            Step := 10;  
        END_IF

    10:

            fbFileOpen(
                sNetId := '', 
                sPathName := sPath, 
                nMode := FOPEN_MODEAPPEND OR FOPEN_MODETEXT, 
                ePath := PATH_GENERIC, 
                bExecute := TRUE
            );      
        Step := 20;

    20:
        // Czekaj na otwarcie pliku
        fbFileOpen(bExecute := FALSE);
        IF NOT fbFileOpen.bBusy THEN
            IF fbFileOpen.bError THEN
                nErrId := fbFileOpen.nErrId;
                bError := TRUE;
                Step := 500;  
            ELSE
                hFile := fbFileOpen.hFile;
                Step := 300;  
            END_IF
        END_IF 

    300:
        // Zamknij plik
        fbFileClose(
            sNetId := '', 
            hFile := hFile, 
            bExecute := TRUE
        );
        Step := 310;

    310:
        // Czekaj na zamknięcie pliku
        fbFileClose(bExecute := FALSE);
        IF NOT fbFileClose.bBusy THEN
            IF fbFileClose.bError THEN
                nErrId := fbFileClose.nErrId;
                bError := TRUE;
            END_IF
            Step := 500;  
        END_IF

    500:
        bBusy := FALSE;
        Step := 0;
END_CASE

END_PROGRAM

// ---- POUs/DataLogging/P_OEE_Raport.TcPOU
PROGRAM P_OEE_Raport
// Zmienne pomocnicze
VAR
    sCurrentDate        : STRING(10) := '';  // Przechowuje aktualną datę (np. "2023-10-25")
    bNewDay             : BOOL := FALSE;     // Flaga wskazująca, że rozpoczął się nowy dzień
    hFile               : UINT := 0;        // Uchwyt pliku
    sFilePath           : T_MaxString := ''; // Ścieżka do pliku
    nBytesToWrite       : UDINT := 0;        // Liczba bajtów do zapisania
    sLineToWrite             : T_MaxString := ''; // Bufor na dane do zapisania
    dtString            : STRING(20) := '';  // Czas zmiany w formacie tekstowym
    fbFileSeek          : FB_FileSeek;       // Blok do pozycjonowania wskaźnika pliku
    fbFileTell          : FB_FileTell;       // Blok do odczytu pozycji wskaźnika pliku
    fbFileGets          : FB_FileGets;       // Blok do odczytu linii z pliku
    bFileIsEmpty        : BOOL := FALSE;     // Flaga wskazująca, czy plik jest pusty
	RisingEdge			:R_trig;
	bSaveManuel			:BOOL;
	Step				:INT;
	bBusy 				:BOOL;
	bError				:BOOL;
	nErrId				:UDINT;
	nIndex				:INT;
	sFolderPath: STRING(255) := 'C:\OEE\';
	fbFileOpen: FB_FileOpen;
    fbFileWrite: FB_FileWrite;
    fbFileClose: FB_FileClose;
	b10step:BOOL;
	rtrig10MinsWork :r_trig;
	tonworkfor10min	:TON;
	AStBadPackageReasonText :ARRAY[0..63] OF S_Information_Text;
    i : INT;
    aIdToName: ARRAY[11..24] OF WSTRING := [
        "Wadliwa butelka lub proces przerwany:","Waga za mała:","Waga za duża:",
        "Brak odłożenia platynki:", "Platynka źle położona:", "Platynka nie zgrzana:",
        "Brak nas.(Słomka):", "Brak nasadki za zakręcarkami:","Brak nasadki przed zakręcarką:",
        "Nie zakręcono zakręcarką szczękową:", "Nasadka źle zakręcona:", "ROPP nie nałożony", 
		"ROPP nie zakręcony","ROPP brak za stacją"];
	bWork10min: BOOL;
	tontimerforevery10min :ton;
END_VAR

// Główna logika
IF Step=0 THEN
	bError:=FALSE;
END_IF
rtrig10MinsWork(CLK:=P_ADS_OEE.btonDelayAfterStart);
tonworkfor10min(in:=bWork10min, PT:=T#5M);
tontimerforevery10min(in:=NOT bWork10min AND P_ADS_OEE.btonDelayAfterStart, PT:=T#5M);
IF rtrig10MinsWork.Q  OR bSaveManuel OR tontimerforevery10min.q THEN
	bWork10min:=TRUE;
END_IF
IF tonworkfor10min.Q THEN
	bWork10min:=FALSE;
END_IF
RisingEdge(CLK := bSaveManuel OR tonworkfor10min.q OR P_ADS_OEE.bCycleReset OR P_ADS_OEE.btonConfectionEnding);

IF rtrig10MinsWork.Q  OR RisingEdge.q THEN 
	FOR i := 0 TO 63 DO
	    IF (P_ADS_OEE.AStBadPackageReason[i].udiID >= 11) AND (P_ADS_OEE.AStBadPackageReason[i].udiID <= 24) THEN
	        AStBadPackageReasonText[i].desc := aIdToName[P_ADS_OEE.AStBadPackageReason[i].udiID];
	    ELSE
	        AStBadPackageReasonText[i].desc := "";
	    END_IF;
	   
	    AStBadPackageReasonText[i].wsDescription := P_ADS_OEE.AStBadPackageReason[i].wsDescription;
	END_FOR;
END_IF

CASE Step OF
    0:
        // Sprawdź, czy zmienił się dzień
        IF LEFT(WSTRING_TO_STRING(P_time.s_time_mainscreen), 10) <> sCurrentDate THEN
            sCurrentDate := LEFT(WSTRING_TO_STRING(P_time.s_time_mainscreen), 10);  // Zaktualizuj datę
            bNewDay := TRUE;  // Ustaw flagę nowego dnia
        END_IF

        // Jeśli wystąpiło zdarzenie zapisu lub zmiany receptury
        IF RisingEdge.Q THEN
            bBusy := TRUE;
            bError := FALSE;
            nErrId := 0;
            nIndex := 0;

            // Utwórz ścieżkę do pliku na podstawie aktualnej daty
            sFilePath := CONCAT(sFolderPath, 'OEE_Raport_');
            sFilePath := CONCAT(sFilePath, sCurrentDate);
            sFilePath := CONCAT(sFilePath, '.csv');

            Step := 10;  // Przejdź do kroku otwarcia pliku
        END_IF

    10:
        // Otwórz plik
        IF bNewDay THEN
            // Jeśli nowy dzień, otwórz plik w trybie zapisu (tworzy nowy plik)
            fbFileOpen(
                sNetId := '', 
                sPathName := sFilePath, 
                nMode := FOPEN_MODEWRITE OR FOPEN_MODETEXT, 
                ePath := PATH_GENERIC, 
                bExecute := TRUE
            );
            b10step := TRUE;
        ELSE
            // Jeśli stary dzień, otwórz plik w trybie dopisywania
            fbFileOpen(
                sNetId := '', 
                sPathName := sFilePath, 
                nMode := FOPEN_MODEAPPEND OR FOPEN_MODETEXT, 
                ePath := PATH_GENERIC, 
                bExecute := TRUE
            );
            b10step := TRUE;
        END_IF
        Step := 20;

    20:
        // Czekaj na otwarcie pliku
        fbFileOpen(bExecute := FALSE);
        IF NOT fbFileOpen.bBusy THEN
            IF fbFileOpen.bError THEN
                nErrId := fbFileOpen.nErrId;
                bError := TRUE;
                Step := 500;  // Przejdź do kroku obsługi błędów
            ELSE
                hFile := fbFileOpen.hFile;
                Step := 30;  // Przejdź do kroku weryfikacji pliku
            END_IF
        END_IF

    30:
        // Sprawdź, czy plik jest pusty (tylko dla nowego dnia)
        IF bNewDay THEN
            fbFileTell(
                sNetId := '', 
                hFile := hFile, 
                bExecute := TRUE
            );
            Step := 35;
        ELSE
            Step := 40;  // Pomijaj weryfikację dla starego dnia
        END_IF

    35:
        // Czekaj na odczyt pozycji wskaźnika pliku
        fbFileTell(bExecute := FALSE);
        IF NOT fbFileTell.bBusy THEN
            IF fbFileTell.nSeekPos = 0 THEN
                bFileIsEmpty := TRUE;  // Plik jest pusty
            ELSE
                bFileIsEmpty := FALSE; // Plik nie jest pusty
            END_IF
            Step := 40;
        END_IF

    40:
        // Przygotuj dane do zapisu
        IF NOT fbFileTell.bBusy THEN
            sLineToWrite := CONCAT(WSTRING_TO_STRING(P_time.s_time_mainscreen), '|');
			sLineToWrite := CONCAT(sLineToWrite, WSTRING_TO_STRING(gvl_recipe.s_recipe_name));
            sLineToWrite := CONCAT(sLineToWrite, '|');
			sLineToWrite := CONCAT(sLineToWrite, INT_TO_STRING(REAL_TO_INT(P_ADS_OEE.uiCounterBadBottles)));
			sLineToWrite := CONCAT(sLineToWrite, '|');
            sLineToWrite := CONCAT(sLineToWrite, INT_TO_STRING(REAL_TO_INT(P_ADS_OEE.uiCounterGoodBottles)));
			sLineToWrite := CONCAT(sLineToWrite, '|');
			sLineToWrite := CONCAT(sLineToWrite, WSTRING_TO_STRING(AStBadPackageReasonText[0].desc));
            sLineToWrite := CONCAT(sLineToWrite, ':');
            sLineToWrite := CONCAT(sLineToWrite, WSTRING_TO_STRING(AStBadPackageReasonText[0].wsDescription));
			sLineToWrite := CONCAT(sLineToWrite, '|');			
            sLineToWrite := CONCAT(sLineToWrite, WSTRING_TO_STRING(AStBadPackageReasonText[1].desc));
            sLineToWrite := CONCAT(sLineToWrite, ':');
            sLineToWrite := CONCAT(sLineToWrite, WSTRING_TO_STRING(AStBadPackageReasonText[1].wsDescription));
			sLineToWrite := CONCAT(sLineToWrite, '|');
			sLineToWrite := CONCAT(sLineToWrite, WSTRING_TO_STRING(AStBadPackageReasonText[2].desc));
            sLineToWrite := CONCAT(sLineToWrite, ':');                                     
            sLineToWrite := CONCAT(sLineToWrite, WSTRING_TO_STRING(AStBadPackageReasonText[2].wsDescription));
			sLineToWrite := CONCAT(sLineToWrite, '|');
			sLineToWrite := CONCAT(sLineToWrite, WSTRING_TO_STRING(AStBadPackageReasonText[3].desc));
            sLineToWrite := CONCAT(sLineToWrite, ':');
            sLineToWrite := CONCAT(sLineToWrite, WSTRING_TO_STRING(AStBadPackageReasonText[3].wsDescription));
			sLineToWrite := CONCAT(sLineToWrite, '|');
			sLineToWrite := CONCAT(sLineToWrite, WSTRING_TO_STRING(AStBadPackageReasonText[4].desc));
            sLineToWrite := CONCAT(sLineToWrite, ':');
            sLineToWrite := CONCAT(sLineToWrite, WSTRING_TO_STRING(AStBadPackageReasonText[4].wsDescription));
			sLineToWrite := CONCAT(sLineToWrite, '|');
			sLineToWrite := CONCAT(sLineToWrite, WSTRING_TO_STRING(AStBadPackageReasonText[5].desc));
            sLineToWrite := CONCAT(sLineToWrite, ':');
            sLineToWrite := CONCAT(sLineToWrite, WSTRING_TO_STRING(AStBadPackageReasonText[5].wsDescription));
			sLineToWrite := CONCAT(sLineToWrite, '|');
			sLineToWrite := CONCAT(sLineToWrite, WSTRING_TO_STRING(AStBadPackageReasonText[6].desc));
            sLineToWrite := CONCAT(sLineToWrite, ':');
            sLineToWrite := CONCAT(sLineToWrite, WSTRING_TO_STRING(AStBadPackageReasonText[6].wsDescription));
			sLineToWrite := CONCAT(sLineToWrite, '|');
			sLineToWrite := CONCAT(sLineToWrite, WSTRING_TO_STRING(AStBadPackageReasonText[7].desc));
            sLineToWrite := CONCAT(sLineToWrite, ':');
            sLineToWrite := CONCAT(sLineToWrite, WSTRING_TO_STRING(AStBadPackageReasonText[7].wsDescription));
			sLineToWrite := CONCAT(sLineToWrite, '|');
			sLineToWrite := CONCAT(sLineToWrite, WSTRING_TO_STRING(AStBadPackageReasonText[8].desc));
            sLineToWrite := CONCAT(sLineToWrite, ':');
            sLineToWrite := CONCAT(sLineToWrite, WSTRING_TO_STRING(AStBadPackageReasonText[8].wsDescription));
			sLineToWrite := CONCAT(sLineToWrite, '|');
			sLineToWrite := CONCAT(sLineToWrite, WSTRING_TO_STRING(AStBadPackageReasonText[9].desc));
            sLineToWrite := CONCAT(sLineToWrite, ':');
            sLineToWrite := CONCAT(sLineToWrite, WSTRING_TO_STRING(AStBadPackageReasonText[9].wsDescription));
			sLineToWrite := CONCAT(sLineToWrite, '|');
			sLineToWrite := CONCAT(sLineToWrite, WSTRING_TO_STRING(AStBadPackageReasonText[10].desc));
            sLineToWrite := CONCAT(sLineToWrite, ':');
            sLineToWrite := CONCAT(sLineToWrite, WSTRING_TO_STRING(AStBadPackageReasonText[10].wsDescription));
			sLineToWrite := CONCAT(sLineToWrite, '|');
			sLineToWrite := CONCAT(sLineToWrite, WSTRING_TO_STRING(AStBadPackageReasonText[11].desc));
            sLineToWrite := CONCAT(sLineToWrite, ':');
            sLineToWrite := CONCAT(sLineToWrite, WSTRING_TO_STRING(AStBadPackageReasonText[11].wsDescription));
			sLineToWrite := CONCAT(sLineToWrite, '|');
			sLineToWrite := CONCAT(sLineToWrite, WSTRING_TO_STRING(AStBadPackageReasonText[12].desc));
            sLineToWrite := CONCAT(sLineToWrite, ':');
            sLineToWrite := CONCAT(sLineToWrite, WSTRING_TO_STRING(AStBadPackageReasonText[12].wsDescription));
			sLineToWrite := CONCAT(sLineToWrite, '|');
			sLineToWrite := CONCAT(sLineToWrite, WSTRING_TO_STRING(AStBadPackageReasonText[13].desc));
            sLineToWrite := CONCAT(sLineToWrite, ':');
            sLineToWrite := CONCAT(sLineToWrite, WSTRING_TO_STRING(AStBadPackageReasonText[13].wsDescription));
			sLineToWrite := CONCAT(sLineToWrite, '|');
			sLineToWrite := CONCAT(sLineToWrite, 'Czas pracy(min):');
			sLineToWrite := CONCAT(sLineToWrite, UINT_TO_STRING(P_ADS_OEE.udiCounterExecuteTime));
			sLineToWrite := CONCAT(sLineToWrite, '$N');

            nBytesToWrite := LEN(sLineToWrite);

            // Zapisz dane do pliku
            fbFileWrite(
                sNetId := '', 
                hFile := hFile, 
                pWriteBuff := ADR(sLineToWrite), 
                cbWriteLen := nBytesToWrite, 
                bExecute := TRUE
            );
            Step := 50;
        ELSE
            Step := 300;  // Przejdź do kroku zamknięcia pliku
        END_IF

    50:
        // Czekaj na zakończenie zapisu
        fbFileWrite(bExecute := FALSE);
        IF NOT fbFileWrite.bBusy THEN
            IF fbFileWrite.bError THEN
                nErrId := fbFileWrite.nErrId;
                bError := TRUE;
                Step := 500;  // Przejdź do kroku obsługi błędów
            ELSE
                Step := 300;  // Przejdź do kroku zamknięcia pliku po jednokrotnym zapisie
            END_IF
        END_IF

    300:
        // Zamknij plik
        fbFileClose(
            sNetId := '', 
            hFile := hFile, 
            bExecute := TRUE
        );
        Step := 310;

    310:
        // Czekaj na zamknięcie pliku
        fbFileClose(bExecute := FALSE);
        IF NOT fbFileClose.bBusy THEN
            IF fbFileClose.bError THEN
                nErrId := fbFileClose.nErrId;
                bError := TRUE;
            END_IF
            Step := 500;  // Przejdź do kroku obsługi błędów
        END_IF

    500:
        // Zakończ procedurę
        bBusy := FALSE;
        bNewDay := FALSE;  // Zresetuj flagę nowego dnia
        Step := 0;
END_CASE

END_PROGRAM

// ---- POUs/ADS/P_ADS_OEE.TcPOU
PROGRAM P_ADS_OEE
VAR
	btonDelayAfterStart :BOOL;
	fbRead_1: FB_ReadAdsSymByName;	
	fbCyclicReadout: TON;
	uiCounterGoodBottles :UINT;
	fbRead_2: FB_ReadAdsSymByName;
	AStBadPackageReason  :ARRAY[0..63] OF S_Information;
	fbRead_3: FB_ReadAdsSymByName;
	uiCounterBadBottles  :UINT;
	fbRead_4: FB_ReadAdsSymByName;
	fbRead_5: FB_ReadAdsSymByName;
	bCycleReset :BOOL;
	udiCounterExecuteTime :UINT;
	fbRead_6: FB_ReadAdsSymByName;
	btonConfectionEnding:BOOL;
	fbRead_7: FB_ReadAdsSymByName;
	
END_VAR

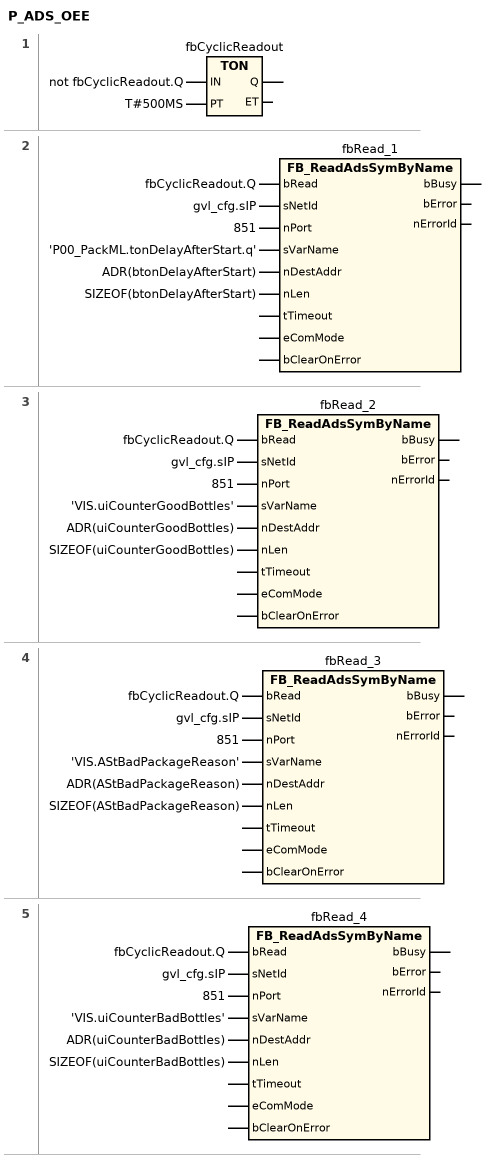
// NETWORK 1
fbCyclicReadout(IN := not fbCyclicReadout.Q, PT := T#500MS); // TON

// NETWORK 2
fbRead_1(
    bRead := fbCyclicReadout.Q,
    sNetId := gvl_cfg.sIP,
    nPort := 851,
    sVarName := 'P00_PackML.tonDelayAfterStart.q',
    nDestAddr := ADR(btonDelayAfterStart),
    nLen := SIZEOF(btonDelayAfterStart)); // FB_ReadAdsSymByName

// NETWORK 3
fbRead_2(
    bRead := fbCyclicReadout.Q,
    sNetId := gvl_cfg.sIP,
    nPort := 851,
    sVarName := 'VIS.uiCounterGoodBottles',
    nDestAddr := ADR(uiCounterGoodBottles),
    nLen := SIZEOF(uiCounterGoodBottles)); // FB_ReadAdsSymByName

// NETWORK 4
fbRead_3(
    bRead := fbCyclicReadout.Q,
    sNetId := gvl_cfg.sIP,
    nPort := 851,
    sVarName := 'VIS.AStBadPackageReason',
    nDestAddr := ADR(AStBadPackageReason),
    nLen := SIZEOF(AStBadPackageReason)); // FB_ReadAdsSymByName

// NETWORK 5
fbRead_4(
    bRead := fbCyclicReadout.Q,
    sNetId := gvl_cfg.sIP,
    nPort := 851,
    sVarName := 'VIS.uiCounterBadBottles',
    nDestAddr := ADR(uiCounterBadBottles),
    nLen := SIZEOF(uiCounterBadBottles)); // FB_ReadAdsSymByName

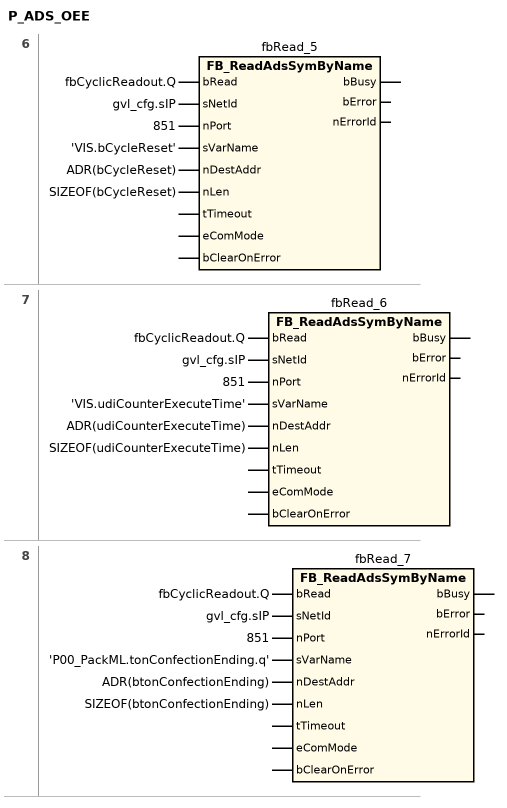
// NETWORK 6
fbRead_5(
    bRead := fbCyclicReadout.Q,
    sNetId := gvl_cfg.sIP,
    nPort := 851,
    sVarName := 'VIS.bCycleReset',
    nDestAddr := ADR(bCycleReset),
    nLen := SIZEOF(bCycleReset)); // FB_ReadAdsSymByName

// NETWORK 7
fbRead_6(
    bRead := fbCyclicReadout.Q,
    sNetId := gvl_cfg.sIP,
    nPort := 851,
    sVarName := 'VIS.udiCounterExecuteTime',
    nDestAddr := ADR(udiCounterExecuteTime),
    nLen := SIZEOF(udiCounterExecuteTime)); // FB_ReadAdsSymByName

// NETWORK 8
fbRead_7(
    bRead := fbCyclicReadout.Q,
    sNetId := gvl_cfg.sIP,
    nPort := 851,
    sVarName := 'P00_PackML.tonConfectionEnding.q',
    nDestAddr := ADR(btonConfectionEnding),
    nLen := SIZEOF(btonConfectionEnding)); // FB_ReadAdsSymByName

END_PROGRAM

// ---- POUs/Persistent/P_PersistentDataSave.TcPOU
PROGRAM P_PersistentDataSave
VAR
	fbSaveChanges :FB_Save;
	sFolderPath: STRING(255) := 'C:\Recipe_changes\';
END_VAR

IF P_persistent.bWritePersistent THEN
	fbSaveChanges.sFilePath := CONCAT(sFolderPath, 'Recipe_change');
    fbSaveChanges.sFilePath := CONCAT(fbSaveChanges.sFilePath, p_24h_C1_2.sCurrentDate);
    fbSaveChanges.sFilePath := CONCAT(fbSaveChanges.sFilePath, '.csv');
	fbSaveChanges();
END_IF

END_PROGRAM

// ---- FB/FB_Save.TcPOU
//-----------------------------------------------------------------------------------------------------
//																
//									 	Tkmatik sp z o.o.
//
//	Name					:		FB_Save
//	Author					:		AM
//	Release Date			:		12.01.2022
//	Current ver				:		v 0.1
// 	Last correction 		:		12.01.2022
// 
//	Description				:
//		Special FB for saving structures to BINARY files						
//
//	Requared hardware		:
//
// 	Configuration			:
//
//
//-----------------------------------------------------------------------------------------------------

FUNCTION_BLOCK FB_Save
VAR_INPUT
	sFilePath											:	STRING(255);					//	File path (e.g. 'C:\1.txt'
	pStructAdr											:	PVOID;                          //	Pointer on data struct
	udiStructSize										:	UDINT;                          //	Size of datastruct
	bExecute											:	BOOL;                           //
END_VAR                                                                                     
VAR_OUTPUT                                                                                  
	bBusy												:	BOOL;                           //	FB is Busy
	bDone												:	BOOL;                           //	Load cycle done, DATA actual 
	bError												:	BOOL;                           //	Flag error
	nErrId												:	UDINT;                          //	Error ID
END_VAR                                                                                     
VAR                                                                                         
	fbFileOpen											:	FB_FileOpen;                    //	FB for opening 
	fbFileClose											:	FB_FileClose;                   //	FB for closing
	fbFileWrite											:	FB_FileWrite;                   //	FB for saving
	hFile												:	UINT;                           //	File hendler
	eMainCase											:	E_FileOpSteps;                  //	Main cycle case value
	rtExecute											:	R_TRIG;                         //	Rtrig for start
END_VAR

ACT_FBs();
ACT_Main();

ACTION ACT_FBs:
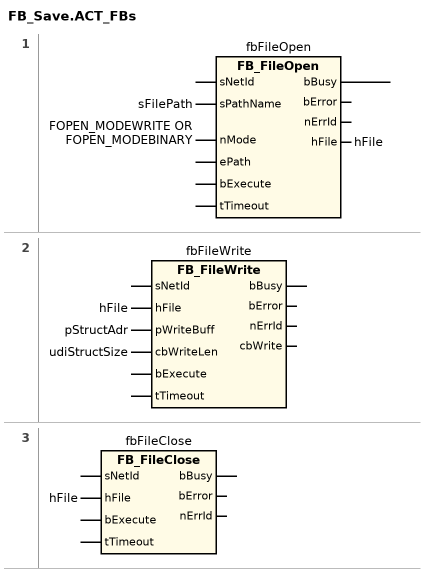
// NETWORK 1
fbFileOpen(sPathName := sFilePath, nMode := FOPEN_MODEWRITE OR FOPEN_MODEBINARY, hFile => hFile); // FB_FileOpen

// NETWORK 2
fbFileWrite(hFile := hFile, pWriteBuff := pStructAdr, cbWriteLen := udiStructSize); // FB_FileWrite

// NETWORK 3
fbFileClose(hFile := hFile); // FB_FileClose
END_ACTION

ACTION ACT_Main:
rtExecute(CLK:=bExecute);
IF (NOT bExecute) THEN
	bDone												:=	FALSE;
END_IF

CASE eMainCase OF
	E_FileOpSteps.eNop:
		fbFileClose.bExecute							:=	FALSE;
		fbFileOpen.bExecute								:=	FALSE;
		fbFileWrite.bExecute							:=	FALSE;
		bBusy											:=	FALSE;
		
		IF (rtExecute.Q) THEN
			bError										:=	FALSE;
			nErrId										:=	0;
			eMainCase									:=	E_FileOpSteps.eStartOpen;
			bBusy										:=	TRUE;
		END_IF
		
	E_FileOpSteps.eStartOpen:
		fbFileOpen.bExecute								:=	TRUE;
		eMainCase										:=	E_FileOpSteps.eWaitOpen;

	E_FileOpSteps.eWaitOpen:
		IF (fbFileOpen.bError) THEN
			bError										:=	TRUE;
			nErrId										:=	10;
			eMainCase									:=	E_FileOpSteps.eNop;
		END_IF
		IF (NOT fbFileOpen.bBusy) THEN
			fbFileOpen.bExecute							:=	FALSE;
			eMainCase									:=	E_FileOpSteps.eStartOper;
		END_IF
		
	E_FileOpSteps.eStartOper:
		fbFileWrite.bExecute							:=	TRUE;
		eMainCase										:=	E_FileOpSteps.eWaitOper;
		
	E_FileOpSteps.eWaitOper:
		IF (fbFileWrite.bError) THEN
			bError										:=	TRUE;
			nErrId										:=	20;
			eMainCase									:=	E_FileOpSteps.eNop;
		END_IF
		IF (NOT fbFileWrite.bBusy) THEN
			fbFileWrite.bExecute						:=	FALSE;
			eMainCase									:=	E_FileOpSteps.eStartClose;
		END_IF
		
	E_FileOpSteps.eStartClose:
		fbFileClose.bExecute							:=	TRUE;
		eMainCase										:=	E_FileOpSteps.eWaitClose;
	
	E_FileOpSteps.eWaitClose:
		IF (fbFileClose.bError) THEN
			bError										:=	TRUE;
			nErrId										:=	30;
			eMainCase									:=	E_FileOpSteps.eNop;
		END_IF
		IF (NOT fbFileClose.bBusy) THEN
			fbFileClose.bExecute						:=	FALSE;
			bDone										:=	TRUE;
			eMainCase									:=	E_FileOpSteps.eNop;
		END_IF	
		
END_CASE
END_ACTION

END_FUNCTION_BLOCK

// ---- POUs/Persistent/P_Persistent.TcPOU
//==================================================================================================
//							Beckhoff Automation Poland
//									25.04.2018
//		Program obslugujacy pamiec nieulotna 
//	v1.4    || TC v 3.1.4026.19		|| - Obsługa UPS
// 	v1.3	|| TC v 3.1.4022.16		|| - Przeniesienie logowania do EvenLogger'a do programu P_SystemDiag_EventLog
// 	v1.2	|| TC v 3.1.4022.0		|| - Dodanie akcji UPS
//	v1.1 	|| TC v 3.1.4020.14 	|| - Dodane wyjscia bOk, bWarning, bError
//	v1.0 	|| TC v 3.1.4020.0 		|| - Pierwsza wersja
//==================================================================================================
PROGRAM P_Persistent
VAR_INPUT
	sAmsNetID_EtherCATMaster	: T_AmsNetId	:= '192.168.40.160.3.1';			// EtherCAT Master AMS Net ID
	bWritePersistent			: BOOL;
	bReset						: BOOL;
END_VAR
VAR_OUTPUT
	bOK							: BOOL 						:= TRUE;				// Brak bledow i ostrzezen
	bWarning					: BOOL;												// Ostrzezenie
	bError						: BOOL;												// Zbiorcza flaga bledow
	udiErrorID					: UDINT;
	sErrorDescription			: WSTRING;
	bWrited						: BOOL;
	bPowerFailDetect			: BOOL;
END_VAR
VAR																			
	iStep						: INT;
	fbWritePersistentData		: FB_WritePersistentData;
	
	//fbUPS						: FB_S_UPS;
	//fbUPS_CB3011				: FB_S_UPS_CB3011;
	//fbUPS_CX51x0				: FB_S_UPS_CX51x0;
	//fbUPS_CX9020_U900			: FB_S_UPS_CX9020_U900;
	//fbUPS_BAPI					: FB_S_UPS_BAPI;
	fbUPS_CU8130				:FB_GetUPSStatus;
	
	//eUpsMode					: E_S_UPS_Mode;
	//eUpsState					: E_S_UPS_State;
	
	
	iNumberOfWrites				: INT;
	rtWritePersistent			: R_TRIG;
END_VAR


ACT_UPS();
ACT_WritePersistent();

fbUPS_CU8130.stStatus.ePowerStatus;
fbUPS_CU8130.stStatus.eBatteryStatus;
fbUPS_CU8130.stStatus.nPowerFailCnt;
fbUPS_CU8130.stStatus.eCommStatus;
IF fbUPS_CU8130.stStatus.ePowerStatus=2 AND NOT bWrited THEN
	bWritePersistent:=TRUE;
ELSE
	bWritePersistent:=FALSE;
END_IF

ACTION ACT_UPS:
//fbUPS_CX9020_U900
//(
//	sNetID							:= sAmsNetID_EtherCATMaster, 
//	iPLCPort						:= 851, 
//	tTimeout						:= DEFAULT_ADS_TIMEOUT, 
//	eUpsMode						:= E_S_UPS_Mode.eSUPS_WrPersistData_Shutdown,
//	ePersistentMode					:= E_PersistentMode.SPDM_2PASS, 
//	tRecoverTime					:= T#10S, 
//	bPowerFailDetect				=> bPowerFailDetect, 
//	eState							=> eUpsState
//);


//fbUPS_CX51x0
//(
//	sNetID							:= sAmsNetID_EtherCATMaster, 
//	iPLCPort						:= 851, 
//	iUPSPort						:= 16#588, 
//	tTimeout						:= DEFAULT_ADS_TIMEOUT, 
//	eUpsMode						:= E_S_UPS_Mode.eSUPS_WrPersistData_Shutdown, 
//	ePersistentMode					:= E_PersistentMode.SPDM_2PASS, 
//	tRecoverTime					:= T#10S, 
//	bPowerFailDetect				=> bPowerFailDetect, 
//	eState							=> eUpsState
//);
fbUPS_CU8130
(	sNetID							:='192.168.40.180.1.1',
	nPort							:=851,
	bEnable							:=TRUE,
	bValid							=>,
	bError	=>,
	nErrId =>,
	stStatus =>,);
END_ACTION

ACTION ACT_WritePersistent:
rtWritePersistent(CLK:= bWritePersistent);


CASE iStep OF

0:
	IF rtWritePersistent.Q THEN
		fbWritePersistentData.PORT												:= _AppInfo.AdsPort;
		fbWritePersistentData.MODE												:= SPDM_2PASS;	
		fbWritePersistentData.START												:= TRUE;
		bWrited																	:= FALSE;
		iStep:= 10;
	END_IF

10:
	IF NOT fbWritePersistentData.BUSY THEN
		IF NOT fbWritePersistentData.ERR THEN
			fbWritePersistentData.START											:= FALSE;
			bWrited																:= TRUE;	
			iNumberOfWrites														:= iNumberOfWrites + 1;
			iStep:= 20;
		END_IF
	END_IF

	IF fbWritePersistentData.ERR THEN
 	
		bWrited																	:= FALSE;
		bError																	:= TRUE;	
		udiErrorID																:= fbWritePersistentData.ERRID;
		sErrorDescription														:= "Błąd zapisu zmiennych PERSISTENT";
		iStep:= 900;
	END_IF
	
20:
	IF NOT bWritePersistent THEN
		iStep:= 0;
	END_IF	
	
900:
	bOK																			:= FALSE;
	
	IF bReset THEN
		fbWritePersistentData.START												:= FALSE;
	END_IF
	IF NOT bReset THEN
		fbWritePersistentData.START												:= TRUE;
	END_IF
	
	
	IF NOT fbWritePersistentData.BUSY THEN
		IF NOT fbWritePersistentData.ERR THEN 
			bOK																	:= TRUE;
			bError																:= FALSE;
			udiErrorID															:= 0;
			sErrorDescription													:= "";
			iStep:= 0;	
		END_IF
	END_IF
	

END_CASE


fbWritePersistentData();
END_ACTION

END_PROGRAM

// ---- FB/FB_Persistent.TcPOU
FUNCTION_BLOCK FB_Persistent

(********************************************************************************************************)
(*								Beckhoff Automation Poland												*)
(* 									FB_Persistent 	v1.5												*)
(* 										20.08.2014														*)
(* 							v1.5 - zmiana minimalnego interwalu zapisu									*)
(* 					Blok funkcyjny zapisujący zmienne typu persistent na karcie CF						*)
(* 						Możliwy zapis na żądanie lub z określoną częstotliwością.  						*)
(* 				Pozostawienie wejscia tInterval bez zmiennej wyłacza funkcję zapisu cyklicznego			*)
(* 							Minimalny czas między zapisem cyklicznym 30s								*)
(* 				Konieczne jest dodanie biblioteki TcUtilities.lib, TcSystem.lib oraz TcBase.lib			*)
(*			 UWAGA: Blok przygotowany dla RunTime 1 port 851 - typowa konfiguracja 						*)
(*______________________________________________________________________________________________________*)

VAR_INPUT
	bWrite					: BOOL;						(*Zapis na rozkaz *)
	tInterval				: TIME:=T#71582M47S295MS;	(*Czestotliwosc zapisu na karte CF*)
END_VAR
VAR_OUTPUT
	bBusy					: BOOL;
	bErr					: BOOL;
	udErrID					: UDINT;
END_VAR
VAR
	fbWritePersistentData	: FB_WritePersistentData; 	(* Blok zapisu *)
	t1						: TON;						(* Timer zapisu *)
	_GETCURTASKINDEX		: GETCURTASKINDEX;			(* Informacja o Tasku *)
	BIndex					: BYTE;						(* Nr tasku *)
END_VAR

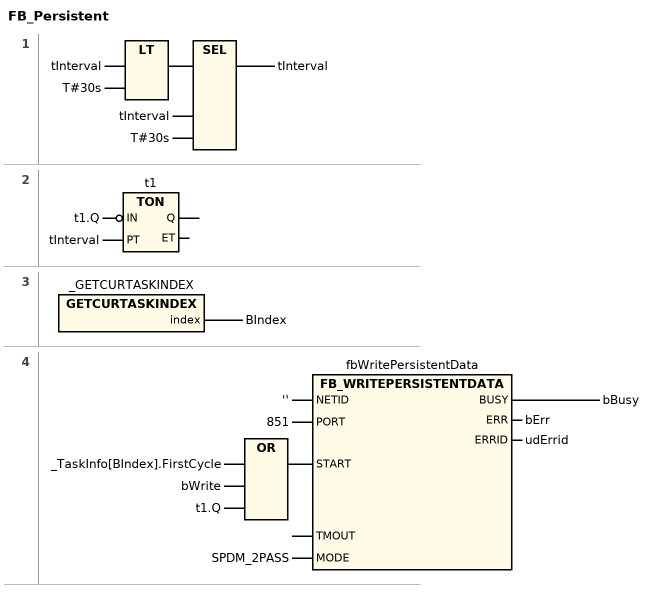
// NETWORK 1
tInterval := SEL(tInterval < T#30s, tInterval, T#30s);

// NETWORK 2
t1(IN := NOT t1.Q, PT := tInterval); // TON

// NETWORK 3
_GETCURTASKINDEX(); // GETCURTASKINDEX
BIndex := _GETCURTASKINDEX.index;

// NETWORK 4
fbWritePersistentData(
    NETID := '',
    PORT := 851,
    START := _TaskInfo[BIndex].FirstCycle OR bWrite OR t1.Q,
    MODE := SPDM_2PASS,
    ERR => bErr,
    ERRID => udErrid); // FB_WRITEPERSISTENTDATA
bBusy := fbWritePersistentData.BUSY;

END_FUNCTION_BLOCK

// ---- FB/FB_ReadWriteLogCSV.TcPOU
(*
Nazwa:			FB_ReadWriteCSV
Opis:			Zapis uzytkownikow do pliku CSV
Wersja:			v0.1
Data:			2018-10-31
Autor:			
Urzadzenia:		
Konfiguracja:	
Info:
*)
FUNCTION_BLOCK FB_ReadWriteLogCSV
VAR
	sCSVLine				: T_MaxString := '';(* Single CSV text line (row, record), we are using string as record buffer (your are able to see read fields)  *)
	sCSVField				: T_MaxString := '';(* Single CSV field value (column, record field) *)
	nRow	 				: UDINT 	:= 0;(* Row number (record) *)
	nColumn					: UDINT 	:= 0;(* Column number (record field) *)
	hFile					: UINT		:= 0;(* File handle of the source file *)
	step					: DWORD 	:= 0;
	fbFileOpen				: FB_FileOpen;(* Opens file *)
	fbFileClose				: FB_FileClose;(* Closes file *)
	fbFileGets				: FB_FileGets;(* Reads one record (line) *)
	fbReader				: FB_CSVMemBufferReader;(* Helper function block used to parse CSV data bytes (single record line) *)
	fbFilePuts				: FB_FilePuts;(* Writes one record (line) *)
	fbWriter				: FB_CSVMemBufferWriter;(* Helper function block used to create CSV data bytes (single record line) *)
	database				: ARRAY[0..239, 0..10] OF STRING(100);(* Target PLC database *)
	i						: INT;
	iNum					: INT;
	BusyFTRIG				: F_TRIG;	// Zakonczenie zapisu/odczytu pliku
	CommandRTRIG			: R_TRIG;	// Wykrycie zapisu/odczytu
	ErrorFileDataUsers		: R_TRIG;	// Błąd zapisu/odczytu
	bNewFile				: BOOL;		// Utworzenie nowego pliku
	iMode					: INT;		// Zapis/odczyt
	
	MAX_CSV_ROWS 			: UDINT := 239;
	MAX_CSV_COLUMNS 		: UDINT := 10;
	MAX_CSV_FIELD_LENGTH	: UDINT := 100;
	
//	fbGetDateTime			: NT_GetTime;
	sDateTime				: STRING[200];
	fbFileTell				: FB_FileTell;
	fbEOF					: FB_EOF;
	fbFileSeek				: FB_FileSeek;
	
	sLineToWrite			:STRING(255);
END_VAR
	
VAR_INPUT
	bRead					: BOOL;		//Sygnal odczytu pliku
	bWrite					: BOOL;		//Sygnal zapisu pliku
	stDataArray				: ARRAY [0..239] OF S_LogData;	//Tablica z danymi
	sNetId					: T_AmsNetId := '';	(* TwinCAT system network address *)
	sFileName				: T_MaxString ;(* CSV destination file path and name *)
END_VAR
VAR_OUTPUT
	bError					: BOOL;		// Sygnal błedu
	bBusy					: BOOL;		// Sygnal zajetosci
	bDone					: BOOL;		// Sygnal zakonczenia odczytu/zapisu
	nErrId					: UDINT;	// Numer bledu
END_VAR

CASE step OF
	0:	(* Wait for rising edge at bWrite variable *)
		IF bWrite (*AND NOT fbGetDateTime.BUSY*) THEN
			bWrite 		:= FALSE;
			bBusy 		:= TRUE;
			bError		:= FALSE;
			nErrId		:= 0;
			hFile		:= 0;
			nRow	 	:= 1;			//było 0
			nColumn		:= 0;
			step 		:= 1;
			//wybiera elementy do zapisania
			FOR iNum := 0 TO TO_INT(MAX_CSV_ROWS) DO
//				sDateTime			:=SYSTEMTIME_TO_STRING(fbGetDateTime.TIMESTR);
//				sDateTime			:=DELETE(sDateTime,11,1);	//Usuwa datę
//				sDateTime			:=LEFT(sDateTime,find(sDateTime,'.')-1); //usuwa licznik ms
				    


				//	sLineToWrite := CONCAT(WSTRING_TO_STRING(P_time.s_time_mainscreen), ',');
   		 		//	sLineToWrite := CONCAT(sLineToWrite, REAL_TO_STRING(P_ADS_SCREW.lrGripperScrewer1TorqueCV));
   		 		//	sLineToWrite := CONCAT(sLineToWrite, ',');
   		 		//	sLineToWrite := CONCAT(sLineToWrite, WSTRING_TO_STRING(gvl_recipe.s_recipe_name));
   		 		//	sLineToWrite := CONCAT(sLineToWrite, '$N');	




				database[iNum,0]		:= WSTRING_TO_STRING(P_time.s_time_mainscreen);
				database[iNum,1]		:= REAL_TO_STRING(stDataArray[iNum].arData[0]);
				database[iNum,2]		:= REAL_TO_STRING(stDataArray[iNum].arData[1]);
				database[iNum,3]		:= REAL_TO_STRING(stDataArray[iNum].arData[2]);
				database[iNum,4]		:= REAL_TO_STRING(stDataArray[iNum].arData[3]);
				database[iNum,5]		:= REAL_TO_STRING(stDataArray[iNum].arData[4]);
				database[iNum,6]		:= REAL_TO_STRING(stDataArray[iNum].arData[5]);
				database[iNum,7]		:= REAL_TO_STRING(stDataArray[iNum].arData[6]);
				database[iNum,8]		:= REAL_TO_STRING(stDataArray[iNum].arData[7]);
				database[iNum,9]		:= REAL_TO_STRING(stDataArray[iNum].arData[8]);
				database[iNum,10]		:= REAL_TO_STRING(stDataArray[iNum].arData[9]);
				
//				database[iNum,0]		:= GVL.arLogDataSave1[iNum].tTime;
//				database[iNum,1]		:= REAL_TO_STRING(GVL.arLogDataSave1[iNum].arData[0]);
//				database[iNum,2]		:= REAL_TO_STRING(GVL.arLogDataSave1[iNum].arData[1]);
//				database[iNum,3]		:= REAL_TO_STRING(GVL.arLogDataSave1[iNum].arData[2]);
//				database[iNum,4]		:= REAL_TO_STRING(GVL.arLogDataSave1[iNum].arData[3]);
//				database[iNum,5]		:= REAL_TO_STRING(GVL.arLogDataSave1[iNum].arData[4]);
//				database[iNum,6]		:= REAL_TO_STRING(GVL.arLogDataSave1[iNum].arData[5]);
//				database[iNum,7]		:= REAL_TO_STRING(GVL.arLogDataSave1[iNum].arData[6]);
//				database[iNum,8]		:= REAL_TO_STRING(GVL.arLogDataSave1[iNum].arData[7]);
//				database[iNum,9]		:= REAL_TO_STRING(GVL.arLogDataSave1[iNum].arData[8]);
//				database[iNum,10]		:= REAL_TO_STRING(GVL.arLogDataSave1[iNum].arData[9]);
			END_FOR
			//zmienia . na , żeby szybciej przetwarzać dane w excelu
//			FOR i:=1 TO UDINT_TO_INT(MAX_CSV_COLUMNS) BY 1 DO
//				database[1,i]:=REPLACE(database[1,i],',',1,FIND(database[1,i],'.'));
//			END_FOR
		END_IF
	1:	(* Open source file *)
		fbFileOpen(bExecute := FALSE);
		fbFiletell(bExecute := FALSE);	//potrzebne do wykrycia nowego pliku
	//	fbEOF(bExecute:=FALSE);
		fbFileSeek(bExecute:=FALSE);	//potrzebne do wykrycia nowego pliku
		fbFileOpen( 	sNetId := sNetId, sPathName := sFileName, nMode := FOPEN_MODEAPPEND OR FOPEN_MODETEXT,(* Open file in TEXT mode! *)
						ePath := PATH_GENERIC, bExecute := TRUE );
		step := 2;
	2:(* Wait until open not busy *)
		fbFileOpen( bExecute := FALSE, bError => bError, nErrID => nErrID, hFile => hFile );
		
		IF NOT fbFileOpen.bBusy THEN
			IF NOT fbFileOpen.bError THEN
				//step := 3;
				//sprawdź czy to nowy plik czy dopisujesz
				//próbuje cofnąć pointer odczytu o -2
				fbFileSeek(sNetId := sNetId,eOrigin := SEEK_END, nSeekPos:=-2, hFile := hFile, bExecute:= TRUE, tTimeout:=T#2S);
				IF NOT fbFileSeek.bBusy THEN
					//sprawdzam gdzie jest pointer
					fbFileTell(sNetId := sNetId, hFile := hFile, bExecute:= TRUE, tTimeout:=T#2S);
					IF NOT fbFileTell.bBusy THEN
						step := 3;
						//jak pointer = 0 to znaczy że zapisano nowy plik - dodaj nagłówki do Excela
						IF fbFileTell.nSeekPos = 0 THEN
							database[1,0]		:='Czas';
							database[1,1]		:= GVL_Screw.arDataLogScrew[0];
							database[1,2]		:= GVL_Screw.arDataLogScrew[1];
							database[1,3]		:= GVL_Screw.arDataLogScrew[2];
							database[1,4]		:= GVL_Screw.arDataLogScrew[3];
							database[1,5]		:= GVL_Screw.arDataLogScrew[4];
							database[1,6]		:= GVL_Screw.arDataLogScrew[5];
							database[1,7]		:= GVL_Screw.arDataLogScrew[6];
							database[1,8]		:= GVL_Screw.arDataLogScrew[7];
							database[1,9]		:= GVL_Screw.arDataLogScrew[8];
							database[1,10]		:= GVL_Screw.arDataLogScrew[9];
						END_IF
					END_IF
				END_IF
			ELSE(* Error: file not found? *)
				step := 100;
			END_IF
		END_IF
	3:(* Convert one PLC record to CSV format *)
		sCSVLine := '';
		fbWriter.eCmd := eEnumCmd_First;(* Write first field value *)
		IF nRow <= MAX_CSV_ROWS THEN
			FOR nColumn := 0 TO MAX_CSV_COLUMNS BY 1 DO
				sCSVField := STRING_TO_CSVFIELD( database[ nRow, nColumn ], FALSE );(* TODO: Get field value from your application *)
				(* Add new field to the record buffer *)
				fbWriter( 	pBuffer := ADR( sCSVLine ), cbBuffer := SIZEOF( sCSVLine ) - 1, putValue := sCSVField, pValue := 0, cbValue := 0,
							bCRLF := ( nColumn = MAX_CSV_COLUMNS ) );(* bCRLF == TRUE => Write CRLF after the last field value *)
				IF fbWriter.bOk THEN
					fbWriter.eCmd := eEnumCmd_Next;(* Write next field value *)
				ELSE(* Error *)
					step := 100;
					RETURN;
				END_IF
			END_FOR(* FOR nColumn := 0... *)
			(* FB_FilePuts adds allready CR (carriage return) to the written line.
			We have to replace the $R$L characters with $L character to avoid double CR. *)
			IF RIGHT( sCSVLine, 2 ) = '$R$L' THEN
				sCSVLine := REPLACE( sCSVLine, '$L', 2, LEN( sCSVLine ) - 1 );
			END_IF
			nRow := nRow + 1;(* Increment number of created records (rows) *)
			step := 4;(* Write record to the file *)
		ELSE(* All rows written => Close file *)
			step := 10;
		END_IF
	4:	(* Write single text line *)
		fbFilePuts( bExecute := FALSE );
		fbFilePuts( sNetId := sNetId, hFile := hFile, sLine := sCSVLine, bExecute := TRUE );
		step := 5;
	5:(* Wait until write not busy *)
		fbFilePuts( bExecute := FALSE, bError => bError, nErrID => nErrID );
		IF NOT fbFilePuts.bBusy THEN
			IF NOT fbFilePuts.bError THEN
				step := 3;(* Write next record *)
			ELSE(* Error *)
				step := 100;
			END_IF
		END_IF
	10:	(* Close source file *)
		fbFileClose( bExecute := FALSE );
		fbFileClose( sNetId := sNetId, hFile := hFile, bExecute := TRUE );
		step := 11;
	11:(* Wait until close not busy *)
		fbFileClose( bExecute := FALSE, bError => bError, nErrID => nErrID );
		IF ( NOT fbFileClose.bBusy ) THEN
			hFile := 0;
			step := 100;
		END_IF
	100: (* Error or ready step => cleanup *)
		IF ( hFile <> 0 ) THEN
			step := 10; (* Close the source file *)
		ELSE
			bBusy := FALSE;
			step := 0;	(* Ready *)
		END_IF
END_CASE
//bWriteUsers	:=FALSE;

END_FUNCTION_BLOCK

// ---- FB/FB_SaveLineToFile.TcPOU
(****************************************************************************************)
(*							Beckhoff Automation Poland									*)
(*								FB_SaveLineToFile  v2.0									*)
(*									26.06.2014											*)
(*						Blok funkcyjny zapisujacy tekst do pliku						*)
(*______________________________________________________________________________________
	Versions:
		v1.1	05.08.2016	* Przepisana wersja do TwinCat3
		v1.0	17.09.2012	* Podstawowa wersja z TwinCat2
________________________________________________________________________________________*)
FUNCTION_BLOCK FB_SaveLineToFile
VAR_INPUT
	bExecute	: BOOL;			(* Komenda wpisu *)
	AmsNetId	: T_AmsNetId;	(* AMS NET ID obiektu docelowego, gdy lokalnie, to zmienna moze byc pusta *)
	sPath		: STRING; 		(* Sciezka pliku, np  'Hard Disk\'*)
	sName		: STRING; 		(* Nazwa pliku wraz z rozszerzeniem 'LogFile.txt'; *)
	sLine		: STRING;		(* Tresc wpisu *)
END_VAR
VAR_OUTPUT
	bBusy		: BOOL;
	bError		: BOOL;
END_VAR
VAR
	fbFileOpen	: FB_FileOpen;
	ftOpen		: F_TRIG;
	fbFilePuts	: FB_FilePuts;
	ftPuts		: F_TRIG;
	fbFileClose	: FB_FileClose;
	ftClose		: F_TRIG;
END_VAR
VAR // added by the converter: edge detectors and wires of the graphical bodies
    _w1 : BOOL;
END_VAR

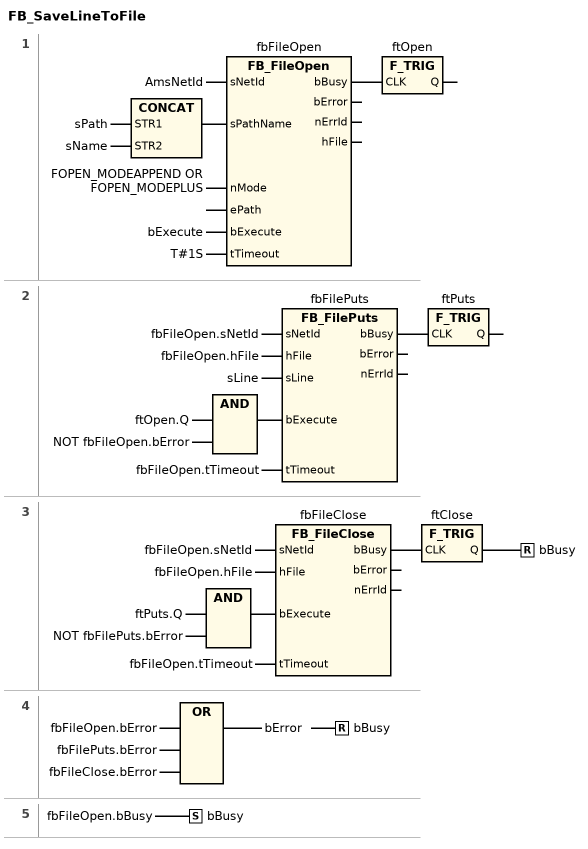
// NETWORK 1
fbFileOpen(
    sNetId := AmsNetId,
    sPathName := CONCAT(STR1 := sPath, STR2 := sName),
    nMode := FOPEN_MODEAPPEND OR FOPEN_MODEPLUS,
    bExecute := bExecute,
    tTimeout := T#1S); // FB_FileOpen
ftOpen(CLK := fbFileOpen.bBusy); // F_TRIG

// NETWORK 2
fbFilePuts(
    sNetId := fbFileOpen.sNetId,
    hFile := fbFileOpen.hFile,
    sLine := sLine,
    bExecute := ftOpen.Q AND (NOT fbFileOpen.bError),
    tTimeout := fbFileOpen.tTimeout); // FB_FilePuts
ftPuts(CLK := fbFilePuts.bBusy); // F_TRIG

// NETWORK 3
fbFileClose(
    sNetId := fbFileOpen.sNetId,
    hFile := fbFileOpen.hFile,
    bExecute := ftPuts.Q AND (NOT fbFilePuts.bError),
    tTimeout := fbFileOpen.tTimeout); // FB_FileClose
ftClose(CLK := fbFileClose.bBusy); // F_TRIG
bBusy R= ftClose.Q;

// NETWORK 4
_w1 := fbFileOpen.bError OR fbFilePuts.bError OR fbFileClose.bError;
bError := _w1;
bBusy R= _w1;

// NETWORK 5
bBusy S= fbFileOpen.bBusy;

END_FUNCTION_BLOCK

// ---- FB/FB_SaveTextToFile.TcPOU
(****************************************************************************************)
(*							Beckhoff Automation Poland									*)
(*								FB_SaveTextToFile  v1.0									*)
(*									26.06.2014											*)
(* Blok funkcyjny zapisujacy tekst do pliku, maksymalna dlugosc wpisu 1000 znakow		*)
(*______________________________________________________________________________________*)
FUNCTION_BLOCK FB_SaveTextToFile
VAR_INPUT
	bExecute		: BOOL;			(* Komenda wpisu *)
	AmsNetId		: T_AmsNetId;	(* AMS NET ID obiektu docelowego, gdy lokalnie, to zmienna moze byc pusta *)
	sPath			: STRING; 		(* Sciezka pliku, np  'Hard Disk\'*)
	sName			: STRING; 		(* Nazwa pliku wraz z rozszerzeniem 'LogFile.txt'; *)
	sLine			: STRING(1000);	(* Tresc wpisu *)
END_VAR
VAR_OUTPUT
	bBusy: 			BOOL;
	bError: 		BOOL;
END_VAR
VAR
	fbFileOpen: 	FB_FileOpen;
	ftOpen: 		F_TRIG;
	fbFilePuts: 	FB_FilePutText;
	ftPuts: 		F_TRIG;
	fbFileClose:	FB_FileClose;
	ftClose: 		F_TRIG;
END_VAR
VAR // added by the converter: edge detectors and wires of the graphical bodies
    _w1 : BOOL;
END_VAR

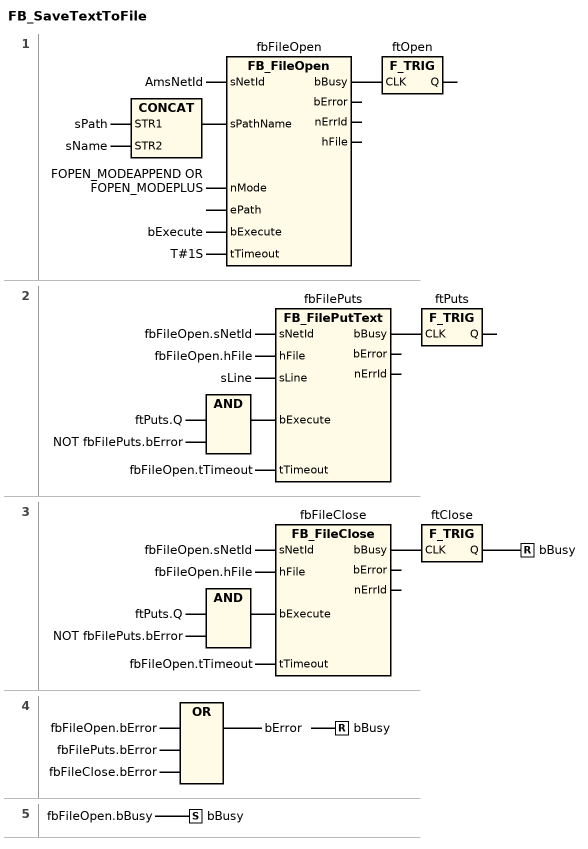
// NETWORK 1
fbFileOpen(
    sNetId := AmsNetId,
    sPathName := CONCAT(STR1 := sPath, STR2 := sName),
    nMode := FOPEN_MODEAPPEND OR FOPEN_MODEPLUS,
    bExecute := bExecute,
    tTimeout := T#1S); // FB_FileOpen
ftOpen(CLK := fbFileOpen.bBusy); // F_TRIG

// NETWORK 2
fbFilePuts(
    sNetId := fbFileOpen.sNetId,
    hFile := fbFileOpen.hFile,
    sLine := sLine,
    bExecute := ftPuts.Q AND (NOT fbFilePuts.bError),
    tTimeout := fbFileOpen.tTimeout); // FB_FilePutText
ftPuts(CLK := fbFilePuts.bBusy); // F_TRIG

// NETWORK 3
fbFileClose(
    sNetId := fbFileOpen.sNetId,
    hFile := fbFileOpen.hFile,
    bExecute := ftPuts.Q AND (NOT fbFilePuts.bError),
    tTimeout := fbFileOpen.tTimeout); // FB_FileClose
ftClose(CLK := fbFileClose.bBusy); // F_TRIG
bBusy R= ftClose.Q;

// NETWORK 4
_w1 := fbFileOpen.bError OR fbFilePuts.bError OR fbFileClose.bError;
bError := _w1;
bBusy R= _w1;

// NETWORK 5
bBusy S= fbFileOpen.bBusy;

END_FUNCTION_BLOCK

// ---- FB/RecipeCSV/FB_ListSaveCSV.TcPOU
//-----------------------------------------------------------------------------------------------------
//																
//									 	Tkmatik sp z o.o.
//
//	Name					:		FB_Save
//	Author					:		AM
//	Release Date			:		12.01.2022
//	Current ver				:		v 0.1
// 	Last correction 		:		12.01.2022
// 
//	Description				:
//		Special FB for saving structures to CSV files						
//
//	Requared hardware		:
//
// 	Configuration			:
//
//
//-----------------------------------------------------------------------------------------------------

FUNCTION_BLOCK FB_ListSaveCSV

VAR_INPUT
	bExecute							: BOOL := FALSE;(* Rising edge starts program execution *)
	sFilePath							: T_MaxString;(* CSV destination file path and name *)
//	database							: POINTER TO STRING(255);	
	nRows          						: UDINT;                // Liczba wierszy
    nCols          						: UDINT; 
	database							: POINTER TO STRING(255);//ARRAY[0..MAX_PARAMS_VARIABLES_COUNT-1] OF STRING(255);
END_VAR
VAR CONSTANT
	MAX_CSV_FIELD_LENGTH				: UDINT	:= 255;	
END_VAR
VAR_IN_OUT
END_VAR

VAR
	
	sNetId			: T_AmsNetId := '';	(* TwinCAT system network address *)
	sCSVLine		: T_MaxString := '';(* Single CSV text line (row, record), we are using string as record buffer (your are able to see created fields) *)
	sCSVField		: T_MaxString := '';(* Single CSV field value (column, record field) *)
	nRow	 		: UDINT 	:= 0;(* Row number (record) *)
	nColumn			: UDINT 	:= 0;(* Column number (record field) *)
	hFile			: UINT		:= 0;(* File handle of the source file *)
	step			: DWORD 	:= 0;
	fbFileOpen		: FB_FileOpen;(* Opens file *)
	fbFileClose		: FB_FileClose;(* Closes file *)
	fbFilePuts		: FB_FilePuts;(* Writes one record (line) *)
	fbWriter		: FB_CSVMemBufferWriter;(* Helper function block used to create CSV data bytes (single record line) *)
	rtExecute		:	R_TRIG;                         //	Rtrig for start



END_VAR
VAR_OUTPUT                                                                                  
	bBusy												:	BOOL;                           //	FB is Busy
	bDone												:	BOOL;                           //	Load cycle done, DATA actual 
	bError												:	BOOL;                           //	Flag error
	nErrId												:	UDINT;                          //	Error ID
END_VAR

rtExecute(CLK:=bExecute);
IF (NOT bExecute) THEN
	bDone												:=	FALSE;
END_IF

CASE step OF
	0:	(* Wait for rising edge at bWrite variable *)
		IF rtExecute.Q THEN
			bBusy 	:= TRUE;
			bError	:= FALSE;
			nErrId	:= 0;
			hFile	:= 0;
			nRow	:= 0;
			nColumn	:= 0;
			step 	:= 1;
		END_IF

	1:	(* Open source file *)
		fbFileOpen(  bExecute := FALSE  );
		fbFileOpen( sNetId := sNetId, sPathName := sFilePath, nMode := FOPEN_MODEWRITE OR FOPEN_MODETEXT,(* Open file in TEXT mode! *)
					ePath := PATH_GENERIC, bExecute := TRUE );
		step := 2;

	2:(* Wait until open not busy *)
		fbFileOpen( bExecute := FALSE, bError => bError, nErrID => nErrID, hFile => hFile );
		IF NOT fbFileOpen.bBusy THEN
			IF NOT fbFileOpen.bError THEN
				step := 3;
			ELSE(* Error: file not found? *)
				step := 100;
			END_IF
		END_IF

	3:(* Convert one PLC record to CSV format *)
		sCSVLine := '';
		fbWriter.eCmd := eEnumCmd_First;(* Write first field value *)
		IF nRow <= nRows THEN

			FOR nColumn := 0 TO nCols BY 1 DO
 
				sCSVField := STRING_TO_CSVFIELD( database[ nRow ], FALSE );(* TODO: Get field value from your application *)

				(* Add new field to the record buffer *)
				fbWriter( 	pBuffer := ADR( sCSVLine ), cbBuffer := SIZEOF( sCSVLine ) - 1, putValue := sCSVField, pValue := 0, cbValue := 0,
							bCRLF := ( nColumn = nCols ) );(* bCRLF == TRUE => Write CRLF after the last field value *)
				IF fbWriter.bOk THEN
					fbWriter.eCmd := eEnumCmd_Next;(* Write next field value *)
				ELSE(* Error *)
					step := 100;
					RETURN;
				END_IF

			END_FOR(* FOR nColumn := 0... *)

			(* FB_FilePuts adds allready CR (carriage return) to the written line.
			We have to replace the $R$L characters with $L character to avoid double CR. *)
			IF RIGHT( sCSVLine, 2 ) = '$R$L' THEN
				sCSVLine := REPLACE( sCSVLine, '$L', 2, LEN( sCSVLine ) - 1 );
			END_IF

			nRow := nRow + 1;(* Increment number of created records (rows) *)
			step := 4;(* Write record to the file *)

		ELSE(* All rows written => Close file *)
			step := 10;
		END_IF

	4:	(* Write single text line *)
		fbFilePuts( bExecute := FALSE );
		fbFilePuts( sNetId := sNetId, hFile := hFile, sLine := sCSVLine, bExecute := TRUE );
		step := 5;

	5:(* Wait until write not busy *)
		fbFilePuts( bExecute := FALSE, bError => bError, nErrID => nErrID );
		IF NOT fbFilePuts.bBusy THEN
			IF NOT fbFilePuts.bError THEN
				step := 3;(* Write next record *)
			ELSE(* Error *)
				step := 100;
			END_IF
		END_IF

	10:	(* Close source file *)
		fbFileClose( bExecute := FALSE );
		fbFileClose( sNetId := sNetId, hFile := hFile, bExecute := TRUE );
		step := 11;

	11:(* Wait until close not busy *)
		fbFileClose( bExecute := FALSE, bError => bError, nErrID => nErrID );
		IF ( NOT fbFileClose.bBusy ) THEN
			bDone	:= TRUE;
			hFile := 0;
			step := 100;
		END_IF

	100: (* Error or ready step => cleanup *)
		IF ( hFile <> 0 ) THEN
			step := 10; (* Close the source file *)
		ELSE
			bBusy := FALSE;
			step := 0;	(* Ready *)
		END_IF

END_CASE

END_FUNCTION_BLOCK

// ---- FB/RecipeCSV/FB_LoadCSV.TcPOU
//-----------------------------------------------------------------------------------------------------
//																
//									 	Tkmatik sp z o.o.
//
//	Name					:		FB_Load
//	Author					:		AM
//	Release Date			:		12.01.2022
//	Current ver				:		v 0.1
// 	Last correction 		:		12.01.2022
// 
//	Description				:
//		Special FB for loading structures from CSV files						
//
//	Requared hardware		:
//
// 	Configuration			:
//
//
//-----------------------------------------------------------------------------------------------------

FUNCTION_BLOCK FB_LoadCSV
VAR_INPUT
	bExecute							: BOOL := FALSE;(* Rising edge starts program execution *)
	sFilePath							: T_MaxString;(* CSV destination file path and name *)
	database							: POINTER TO STRING(255);	
	nRows          						: UDINT;                // Liczba wierszy
    nCols          						: UDINT; 
END_VAR
VAR CONSTANT
	MAX_CSV_FIELD_LENGTH				: UDINT	:= 255;	
END_VAR
VAR_OUTPUT                                                                                  
	bBusy												:	BOOL;                           //	FB is Busy
	bDone												:	BOOL;                           //	Load cycle done, DATA actual 
	bError												:	BOOL;                           //	Flag error
	nErrId												:	UDINT;                          //	Error ID

END_VAR   
VAR_IN_OUT
END_VAR
VAR
	sNetId			: T_AmsNetId := '';	(* TwinCAT system network address *)
	sCSVLine		: T_MaxString := '';(* Single CSV text line (row, record), we are using string as record buffer (your are able to see read fields)  *)
	sCSVField		: T_MaxString := '';(* Single CSV field value (column, record field) *)
	nRow	 		: UDINT 	:= 0;(* Row number (record) *)
	nColumn			: UDINT 	:= 0;(* Column number (record field) *)
	hFile			: UINT		:= 0;(* File handle of the source file *)
	step			: DWORD 	:= 0;
	fbFileOpen		: FB_FileOpen;(* Opens file *)
	fbFileClose		: FB_FileClose;(* Closes file *)
	fbFileGets		: FB_FileGets;(* Reads one record (line) *)
	fbReader		: FB_CSVMemBufferReader;(* Helper function block used to parse CSV data bytes (single record line) *)

//	database		: ARRAY[0..MAX_CSV_ROWS, 0..MAX_CSV_COLUMNS ] OF STRING(MAX_CSV_FIELD_LENGTH);(* Target PLC database *)
	rtExecute		:	R_TRIG;                         //	Rtrig for start
END_VAR

rtExecute(CLK:=bExecute);
IF (NOT bExecute) THEN
	bDone												:=	FALSE;
END_IF
CASE step OF
	0:	(* Wait for rising edge at bRead variable *)
		IF rtExecute.Q THEN
			bBusy 	:= TRUE;
			bError	:= FALSE;
			nErrId	:= 0;
			hFile	:= 0;
			nRow	:= 0;
			nColumn	:= 0;
//			MEMSET( ADR( database ), 0, SIZEOF( database ) );
			step 		:= 1;
		END_IF

	1:	(* Open source file *)
		fbFileOpen(  bExecute := FALSE  );
		fbFileOpen( sNetId := sNetId, sPathName := sFilePath, nMode := FOPEN_MODEREAD OR FOPEN_MODETEXT,(* Open file in TEXT mode! *)
					ePath := PATH_GENERIC, bExecute := TRUE);
		step := 2;

	2:(* Wait until open not busy *)
		fbFileOpen( bExecute := FALSE, bError => bError, nErrID => nErrID, hFile => hFile );
		IF NOT fbFileOpen.bBusy THEN
			IF NOT fbFileOpen.bError THEN
				step := 3;
			ELSE(* Error: file not found? *)
				step := 100;
			END_IF
		END_IF

	3:	(* Read single line (record) *)
		fbFileGets( bExecute := FALSE );
		fbFileGets( sNetId := sNetId, hFile := hFile, bExecute := TRUE );
		step := 4;

	4:(* Wait until read not busy *)
		fbFileGets( bExecute := FALSE, bError => bError, nErrID => nErrID, sLine => sCSVLine );
		IF NOT fbFileGets.bBusy THEN
			IF NOT fbFileGets.bError THEN
				IF fbFileGets.bEOF THEN
					step := 10;(* End of file reached => Close source file *)
				ELSE

					(* FB_FileGets returns text line without the CR (carriage return) character.
					We have to restore the CR character (replace the $L character with $R$L characters) *)
					IF RIGHT( sCSVLine, 1 ) = '$L' THEN
						sCSVLine := REPLACE( sCSVLine, '$R$L', 2, LEN( sCSVLine ) );
					END_IF

					step := 5;
				END_IF
			ELSE(* Error *)
				step := 10;
			END_IF
		END_IF

	5:(* Parse single line (record) *)
		fbReader.eCmd := eEnumCmd_First;(* Read first field value *)
		REPEAT
			fbReader( pBuffer := ADR( sCSVLine ), cbBuffer := SIZEOF( sCSVLine ), getValue => sCSVField );
			IF fbReader.bOk THEN
				fbReader.eCmd := eEnumCmd_Next;(* Read next field value *)

				IF ( nRow <= nRows ) THEN
					IF ( nColumn <= nCols ) THEN
						database[nRow] := CSVFIELD_TO_STRING( sCSVField, FALSE );(* TODO: Save or use the field value in your application *)
					END_IF
				END_IF

				nColumn := nColumn + 1;(* Increment number of read columns *)
				IF fbReader.bCRLF THEN(* CRLF == TRUE => End of reacord reached *)
					nRow 		:= nRow + 1;(* Increment number of read records *)
					nColumn 	:= 0;(* Reset number of columns *)
				END_IF

			ELSE(* Error: End of record reached or all fields read *)
				step := 3;(* Try to read next line *)
			END_IF
		UNTIL NOT fbReader.bOk
		END_REPEAT

	10:	(* Close source file *)
		fbFileClose( bExecute := FALSE);
		fbFileClose( sNetId := sNetId, hFile := hFile, bExecute := TRUE );
		step := 11;

	11:(* Wait until close not busy *)
		fbFileClose( bExecute := FALSE, bError => bError, nErrID => nErrID );
		IF ( NOT fbFileClose.bBusy ) THEN
			bDone	:= TRUE;			
			hFile := 0;
			step := 100;
		END_IF

	100: (* Error or ready step => cleanup *)
		IF ( hFile <> 0 ) THEN
			step := 10; (* Close the source file *)
		ELSE
			bBusy := FALSE;
			step := 0;	(* Ready *)
		END_IF

END_CASE

END_FUNCTION_BLOCK

// ---- FB/RecipeCSV/FB_RecipeSaveCSV.TcPOU
//-----------------------------------------------------------------------------------------------------
//																
//									 	Tkmatik sp z o.o.
//
//	Name					:		FB_Save
//	Author					:		AM
//	Release Date			:		12.01.2022
//	Current ver				:		v 0.1
// 	Last correction 		:		12.01.2022
// 
//	Description				:
//		Special FB for saving structures to CSV files						
//
//	Requared hardware		:
//
// 	Configuration			:
//
//
//-----------------------------------------------------------------------------------------------------

FUNCTION_BLOCK FB_RecipeSaveCSV

VAR_INPUT
	bExecute							: BOOL := FALSE;(* Rising edge starts program execution *)
	sFilePath							: T_MaxString;(* CSV destination file path and name *)
//	database							: POINTER TO STRING(255);	
	nRows          						: UDINT;                // Liczba wierszy
    nCols          						: UDINT; 
	database							: POINTER TO STRING(255);//ARRAY[0..MAX_PARAMS_VARIABLES_COUNT-1] OF STRING(255);
END_VAR
VAR CONSTANT
	MAX_CSV_FIELD_LENGTH				: UDINT	:= 255;	
END_VAR
VAR_IN_OUT
END_VAR

VAR
	
	sNetId			: T_AmsNetId := '';	(* TwinCAT system network address *)
	sCSVLine		: T_MaxString := '';(* Single CSV text line (row, record), we are using string as record buffer (your are able to see created fields) *)
	sCSVField		: T_MaxString := '';(* Single CSV field value (column, record field) *)
	nRow	 		: UDINT 	:= 0;(* Row number (record) *)
	nColumn			: UDINT 	:= 0;(* Column number (record field) *)
	hFile			: UINT		:= 0;(* File handle of the source file *)
	step			: DWORD 	:= 0;
	fbFileOpen		: FB_FileOpen;(* Opens file *)
	fbFileClose		: FB_FileClose;(* Closes file *)
	fbFilePuts		: FB_FilePuts;(* Writes one record (line) *)
	fbWriter		: FB_CSVMemBufferWriter;(* Helper function block used to create CSV data bytes (single record line) *)
	rtExecute		:	R_TRIG;                         //	Rtrig for start



END_VAR
VAR_OUTPUT                                                                                  
	bBusy												:	BOOL;                           //	FB is Busy
	bDone												:	BOOL;                           //	Load cycle done, DATA actual 
	bError												:	BOOL;                           //	Flag error
	nErrId												:	UDINT;                          //	Error ID
END_VAR

rtExecute(CLK:=bExecute);
IF (NOT bExecute) THEN
	bDone												:=	FALSE;
END_IF

CASE step OF
	0:	(* Wait for rising edge at bWrite variable *)
		IF rtExecute.Q THEN
			bBusy 	:= TRUE;
			bError	:= FALSE;
			nErrId	:= 0;
			hFile	:= 0;
			nRow	:= 0;
			nColumn	:= 0;
			step 	:= 1;
		END_IF

	1:	(* Open source file *)
		fbFileOpen(  bExecute := FALSE  );
		fbFileOpen( sNetId := sNetId, sPathName := sFilePath, nMode := FOPEN_MODEWRITE OR FOPEN_MODETEXT,(* Open file in TEXT mode! *)
					ePath := PATH_GENERIC, bExecute := TRUE );
		step := 2;

	2:(* Wait until open not busy *)
		fbFileOpen( bExecute := FALSE, bError => bError, nErrID => nErrID, hFile => hFile );
		IF NOT fbFileOpen.bBusy THEN
			IF NOT fbFileOpen.bError THEN
				step := 3;
			ELSE(* Error: file not found? *)
				step := 100;
			END_IF
		END_IF

	3:(* Convert one PLC record to CSV format *)
		sCSVLine := '';
		fbWriter.eCmd := eEnumCmd_First;(* Write first field value *)
		IF nRow <= nRows THEN

			FOR nColumn := 0 TO nCols BY 1 DO
 
				sCSVField := STRING_TO_CSVFIELD( database[ nRow ], FALSE );(* TODO: Get field value from your application *)

				(* Add new field to the record buffer *)
				fbWriter( 	pBuffer := ADR( sCSVLine ), cbBuffer := SIZEOF( sCSVLine ) - 1, putValue := sCSVField, pValue := 0, cbValue := 0,
							bCRLF := ( nColumn = nCols ) );(* bCRLF == TRUE => Write CRLF after the last field value *)
				IF fbWriter.bOk THEN
					fbWriter.eCmd := eEnumCmd_Next;(* Write next field value *)
				ELSE(* Error *)
					step := 100;
					RETURN;
				END_IF

			END_FOR(* FOR nColumn := 0... *)

			(* FB_FilePuts adds allready CR (carriage return) to the written line.
			We have to replace the $R$L characters with $L character to avoid double CR. *)
			IF RIGHT( sCSVLine, 2 ) = '$R$L' THEN
				sCSVLine := REPLACE( sCSVLine, '$L', 2, LEN( sCSVLine ) - 1 );
			END_IF

			nRow := nRow + 1;(* Increment number of created records (rows) *)
			step := 4;(* Write record to the file *)

		ELSE(* All rows written => Close file *)
			step := 10;
		END_IF

	4:	(* Write single text line *)
		fbFilePuts( bExecute := FALSE );
		fbFilePuts( sNetId := sNetId, hFile := hFile, sLine := sCSVLine, bExecute := TRUE );
		step := 5;

	5:(* Wait until write not busy *)
		fbFilePuts( bExecute := FALSE, bError => bError, nErrID => nErrID );
		IF NOT fbFilePuts.bBusy THEN
			IF NOT fbFilePuts.bError THEN
				step := 3;(* Write next record *)
			ELSE(* Error *)
				step := 100;
			END_IF
		END_IF

	10:	(* Close source file *)
		fbFileClose( bExecute := FALSE );
		fbFileClose( sNetId := sNetId, hFile := hFile, bExecute := TRUE );
		step := 11;

	11:(* Wait until close not busy *)
		fbFileClose( bExecute := FALSE, bError => bError, nErrID => nErrID );
		IF ( NOT fbFileClose.bBusy ) THEN
			bDone	:= TRUE;
			hFile := 0;
			step := 100;
		END_IF

	100: (* Error or ready step => cleanup *)
		IF ( hFile <> 0 ) THEN
			step := 10; (* Close the source file *)
		ELSE
			bBusy := FALSE;
			step := 0;	(* Ready *)
		END_IF

END_CASE

END_FUNCTION_BLOCK

// ---- FB/RecipeCSV/FB_RecipeVariablesSaveCSV.TcPOU
//-----------------------------------------------------------------------------------------------------
//																
//									 	Tkmatik sp z o.o.
//
//	Name					:		FB_Save
//	Author					:		AM
//	Release Date			:		12.01.2022
//	Current ver				:		v 0.1
// 	Last correction 		:		12.01.2022
// 
//	Description				:
//		Special FB for saving structures to CSV files						
//
//	Requared hardware		:
//
// 	Configuration			:
//
//
//-----------------------------------------------------------------------------------------------------

FUNCTION_BLOCK FB_RecipeVariablesSaveCSV

VAR_INPUT
	bExecute							: BOOL := FALSE;(* Rising edge starts program execution *)
	sFilePath							: T_MaxString;(* CSV destination file path and name *)
//	database							: POINTER TO STRING(255);	
	nRows          						: UDINT;                // Liczba wierszy
    nCols          						: UDINT; 
	database							: POINTER TO STRING(255);//ARRAY[0..MAX_PARAMS_VARIABLES_COUNT-1] OF STRING(255);
	
END_VAR
VAR CONSTANT
	MAX_CSV_FIELD_LENGTH				: UDINT	:= 255;	
END_VAR
VAR_IN_OUT
END_VAR

VAR
	
	sNetId			: T_AmsNetId := '';	(* TwinCAT system network address *)
	sCSVLine		: T_MaxString := '';(* Single CSV text line (row, record), we are using string as record buffer (your are able to see created fields) *)
	sCSVField		: T_MaxString := '';(* Single CSV field value (column, record field) *)
	nRow	 		: UDINT 	:= 0;(* Row number (record) *)
	nColumn			: UDINT 	:= 0;(* Column number (record field) *)
	hFile			: UINT		:= 0;(* File handle of the source file *)
	step			: DWORD 	:= 0;
	fbFileOpen		: FB_FileOpen;(* Opens file *)
	fbFileClose		: FB_FileClose;(* Closes file *)
	fbFilePuts		: FB_FilePuts;(* Writes one record (line) *)
	fbWriter		: FB_CSVMemBufferWriter;(* Helper function block used to create CSV data bytes (single record line) *)
	rtExecute		:	R_TRIG;                         //	Rtrig for start



END_VAR
VAR_OUTPUT                                                                                  
	bBusy												:	BOOL;                           //	FB is Busy
	bDone												:	BOOL;                           //	Load cycle done, DATA actual 
	bError												:	BOOL;                           //	Flag error
	nErrId												:	UDINT;                          //	Error ID

END_VAR


rtExecute(CLK:=bExecute);
IF (NOT bExecute) THEN
	bDone												:=	FALSE;
END_IF

CASE step OF
	0:	(* Wait for rising edge at bWrite variable *)
		IF rtExecute.Q THEN
			bBusy 	:= TRUE;
			bError	:= FALSE;
			nErrId	:= 0;
			hFile	:= 0;
			nRow	:= 0;
			nColumn	:= 0;
			step 	:= 1;
		END_IF

	1:	(* Open source file *)
		fbFileOpen(  bExecute := FALSE  );
		fbFileOpen( sNetId := sNetId, sPathName := sFilePath, nMode := FOPEN_MODEWRITE OR FOPEN_MODETEXT,(* Open file in TEXT mode! *)
					ePath := PATH_GENERIC, bExecute := TRUE );
		step := 2;

	2:(* Wait until open not busy *)
		fbFileOpen( bExecute := FALSE, bError => bError, nErrID => nErrID, hFile => hFile );
		IF NOT fbFileOpen.bBusy THEN
			IF NOT fbFileOpen.bError THEN
				step := 3;
			ELSE(* Error: file not found? *)
				step := 100;
			END_IF
		END_IF

	3:(* Convert one PLC record to CSV format *)
		sCSVLine := '';
		fbWriter.eCmd := eEnumCmd_First;(* Write first field value *)
		IF nRow <= nRows THEN

			FOR nColumn := 0 TO nCols BY 1 DO
 
				sCSVField := STRING_TO_CSVFIELD( database[ nRow ], FALSE );(* TODO: Get field value from your application *)

				(* Add new field to the record buffer *)
				fbWriter( 	pBuffer := ADR( sCSVLine ), cbBuffer := SIZEOF( sCSVLine ) - 1, putValue := sCSVField, pValue := 0, cbValue := 0,
							bCRLF := ( nColumn = nCols ) );(* bCRLF == TRUE => Write CRLF after the last field value *)
				IF fbWriter.bOk THEN
					fbWriter.eCmd := eEnumCmd_Next;(* Write next field value *)
				ELSE(* Error *)
					step := 100;
					RETURN;
				END_IF

			END_FOR(* FOR nColumn := 0... *)

			(* FB_FilePuts adds allready CR (carriage return) to the written line.
			We have to replace the $R$L characters with $L character to avoid double CR. *)
			IF RIGHT( sCSVLine, 2 ) = '$R$L' THEN
				sCSVLine := REPLACE( sCSVLine, '$L', 2, LEN( sCSVLine ) - 1 );
			END_IF

			nRow := nRow + 1;(* Increment number of created records (rows) *)
			step := 4;(* Write record to the file *)

		ELSE(* All rows written => Close file *)
			step := 10;
		END_IF

	4:	(* Write single text line *)
		fbFilePuts( bExecute := FALSE );
		fbFilePuts( sNetId := sNetId, hFile := hFile, sLine := sCSVLine, bExecute := TRUE );
		step := 5;

	5:(* Wait until write not busy *)
		fbFilePuts( bExecute := FALSE, bError => bError, nErrID => nErrID );
		IF NOT fbFilePuts.bBusy THEN
			IF NOT fbFilePuts.bError THEN
				step := 3;(* Write next record *)
			ELSE(* Error *)
				step := 100;
			END_IF
		END_IF

	10:	(* Close source file *)
		fbFileClose( bExecute := FALSE );
		fbFileClose( sNetId := sNetId, hFile := hFile, bExecute := TRUE );
		step := 11;

	11:(* Wait until close not busy *)
		fbFileClose( bExecute := FALSE, bError => bError, nErrID => nErrID );
		IF ( NOT fbFileClose.bBusy ) THEN
			bDone	:= TRUE;
			hFile := 0;
			step := 100;
		END_IF

	100: (* Error or ready step => cleanup *)
		IF ( hFile <> 0 ) THEN
			step := 10; (* Close the source file *)
		ELSE
			bBusy := FALSE;
			step := 0;	(* Ready *)
		END_IF

END_CASE

END_FUNCTION_BLOCK

// ---- FB/RecipeList/FB_Load.TcPOU
//-----------------------------------------------------------------------------------------------------
//																
//									 	Tkmatik sp z o.o.
//
//	Name					:		FB_Load
//	Author					:		AM
//	Release Date			:		12.01.2022
//	Current ver				:		v 0.1
// 	Last correction 		:		12.01.2022
// 
//	Description				:
//		Special FB for loading structures from BINARY files						
//
//	Requared hardware		:
//
// 	Configuration			:
//
//
//-----------------------------------------------------------------------------------------------------

FUNCTION_BLOCK FB_Load
VAR_INPUT
	sFilePath											:	STRING(255);					//	File path (e.g. 'C:\1.txt')
	pStructAdr											:	PVOID;                          //	Pointer on data struct
	udiStructSize										:	UDINT;                          //	Size of datastruct
	bExecute											:	BOOL;                           //
END_VAR                                                                                     
VAR_OUTPUT                                                                                  
	bBusy												:	BOOL;                           //	FB is Busy
	bDone												:	BOOL;                           //	Load cycle done, DATA actual 
	bError												:	BOOL;                           //	Flag error
	nErrId												:	UDINT;                          //	Error ID
END_VAR                                                                                     
VAR                                                                                         
	fbFileOpen											:	FB_FileOpen;                    //	FB for opening 
	fbFileClose											:	FB_FileClose;                   //	FB for closing
	fbFileRead											:	FB_FileRead;                    //	FB for reading
	hFile												:	UINT;                           //	File hendler
	eMainCase											:	E_FileOpSteps;                  //	Main cycle case value
	rtExecute											:	R_TRIG;                         //	Rtrig for start
END_VAR

ACT_FBs();
ACT_Main();

ACTION ACT_FBs:
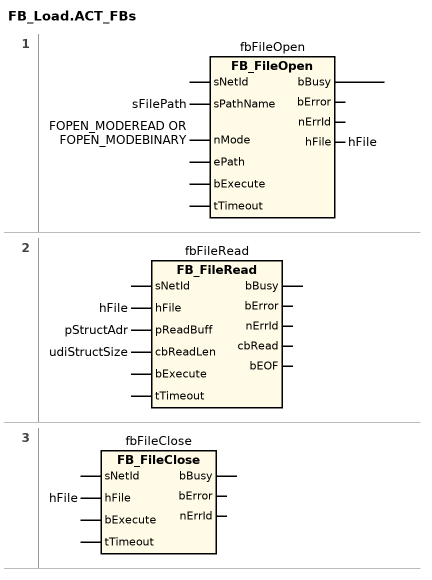
// NETWORK 1
fbFileOpen(sPathName := sFilePath, nMode := FOPEN_MODEREAD OR FOPEN_MODEBINARY, hFile => hFile); // FB_FileOpen

// NETWORK 2
fbFileRead(hFile := hFile, pReadBuff := pStructAdr, cbReadLen := udiStructSize); // FB_FileRead

// NETWORK 3
fbFileClose(hFile := hFile); // FB_FileClose
END_ACTION

ACTION ACT_Main:
rtExecute(CLK:=bExecute);
IF (NOT bExecute) THEN
	bDone												:=	FALSE;
END_IF

CASE eMainCase OF
	E_FileOpSteps.eNop:
		fbFileClose.bExecute							:=	FALSE;
		fbFileOpen.bExecute								:=	FALSE;
		fbFileRead.bExecute								:=	FALSE;
		bBusy											:=	FALSE;
		
		IF (rtExecute.Q) THEN
			bError										:=	FALSE;
			nErrId										:=	0;
			eMainCase									:=	E_FileOpSteps.eStartOpen;
			bBusy										:=	TRUE;
		END_IF
		
	E_FileOpSteps.eStartOpen:
		fbFileOpen.bExecute								:=	TRUE;
		eMainCase										:=	E_FileOpSteps.eWaitOpen;

	E_FileOpSteps.eWaitOpen:
		IF (fbFileOpen.bError) THEN
			bError										:=	TRUE;
			nErrId										:=	10;
			eMainCase									:=	E_FileOpSteps.eNop;
		ELSIF (NOT fbFileOpen.bBusy) THEN
			fbFileOpen.bExecute							:=	FALSE;
			eMainCase									:=	E_FileOpSteps.eStartOper;
		END_IF
		
	E_FileOpSteps.eStartOper:
		fbFileRead.bExecute								:=	TRUE;
		eMainCase										:=	E_FileOpSteps.eWaitOper;
		
	E_FileOpSteps.eWaitOper:
		IF (fbFileRead.bError) THEN
			bError										:=	TRUE;
			nErrId										:=	20;
			eMainCase									:=	E_FileOpSteps.eNop;
		ELSIF (NOT fbFileRead.bBusy) THEN
			fbFileRead.bExecute							:=	FALSE;
			eMainCase									:=	E_FileOpSteps.eStartClose;
		END_IF
		
	E_FileOpSteps.eStartClose:
		fbFileClose.bExecute							:=	TRUE;
		eMainCase										:=	E_FileOpSteps.eWaitClose;
	
	E_FileOpSteps.eWaitClose:
		IF (fbFileClose.bError) THEN
			bError										:=	TRUE;
			nErrId										:=	30;
			eMainCase									:=	E_FileOpSteps.eNop;
		ELSIF (NOT fbFileClose.bBusy) THEN
			fbFileClose.bExecute						:=	FALSE;
			bDone										:=	TRUE;
			eMainCase									:=	E_FileOpSteps.eNop;
		END_IF	
		
END_CASE
END_ACTION

END_FUNCTION_BLOCK

// ---- NotUsedPOU/P_50_screw.TcPOU
PROGRAM P_50_screw
VAR

    fbFileOpen: FB_FileOpen;
    fbFileRead: FB_FileRead;
    fbFileClose: FB_FileClose;
    hFile: UINT;
    sFilePath: STRING(255);
    sBuffer: STRING(1000);
    nBytesRead: UDINT;
    bFileOpen: BOOL := FALSE;
    bFileRead: BOOL := FALSE;
    bFileClose: BOOL := FALSE;
	i:UDINT;
	sParse: STRING:='$N';
    sNumber:STRING(10);
    nNumberIndex: INT := 1; 
    nFileCounter: INT := 1;
    nRowCounter: INT := 1;
    nColCounter: INT := 1;
	cCurrentChar: BYTE;
    sCurrentChar: STRING(1);

    bBusy: BOOL := FALSE;
    bError: BOOL := FALSE;
    nErrId: UDINT;


    sFolderPath: STRING(255) := 'C:\LastScrewingCycles\';
    sFileName: STRING(255);
    sSearchPattern: STRING(255) := 'Zakrecarki_1_*.csv';
    nFileIndex: INT := 1;
END_VAR



(*
IF gvl_screw.bExport AND NOT bBusy THEN
    bBusy := TRUE;
    bError := FALSE;
    nFileCounter := 1;
    nRowCounter := 1;
    nColCounter := 1;


    
    WHILE nFileCounter <= 50 DO
        sFilePath := CONCAT('Zakrecarka_1_', INT_TO_STRING(nFileCounter));
		sFilePath:=Concat(sFilePath,'.csv');
 		sFileName := CONCAT(sFolderPath, sFilePath);
        fbFileOpen(sNetId := '', sPathName := sFileName, nMode := FOPEN_MODEREAD OR FOPEN_MODETEXT, ePath := PATH_GENERIC, bExecute := TRUE);
        IF NOT fbFileOpen.bBusy THEN
            IF fbFileOpen.bError THEN
                bError := TRUE;
                nErrId := fbFileOpen.nErrId;
                EXIT;
            ELSE
                hFile := fbFileOpen.hFile;
                bFileOpen := TRUE;

       
                WHILE TRUE DO
                    fbFileRead(sNetId := '', hFile := hFile, pReadBuff := ADR(sBuffer), cbReadLen := SIZEOF(sBuffer), bExecute := TRUE);
                    IF NOT fbFileRead.bBusy THEN
                        IF fbFileRead.bError THEN
                            bError := TRUE;
                            nErrId := fbFileRead.nErrId;
                            EXIT;
                        ELSE
                            nBytesRead := fbFileRead.cbRead;
                            IF nBytesRead = 0 THEN
                                EXIT; 
                            ELSE
								FOR i := 1 TO nBytesRead DO
								    cCurrentChar := sBuffer[i];
								    sCurrentChar := BYTE_TO_STRING(cCurrentChar); 
								
								    IF sCurrentChar = sParse THEN
								    
								        IF sNumber <> '' THEN
								            gvl_screw.aLast50Screw[nFileCounter, nRowCounter] := STRING_TO_INT(sNumber);
								            nRowCounter := nRowCounter + 1;
								            nColCounter := 1;
								            sNumber := ''; 
								            nNumberIndex := 1;
								        END_IF;
								    ELSE
								        
								        sNumber := CONCAT(sNumber, sCurrentChar);
								    END_IF;
								END_FOR;
                            END_IF;
                        END_IF;
                    END_IF;
                END_WHILE;

        
                fbFileClose(sNetId := '', hFile := hFile, bExecute := TRUE);
                IF NOT fbFileClose.bBusy THEN
                    IF fbFileClose.bError THEN
                        bError := TRUE;
                        nErrId := fbFileClose.nErrId;
                    END_IF;
                    bFileOpen := FALSE;
                END_IF;
            END_IF;
        END_IF;

        nFileCounter := nFileCounter + 1;
    END_WHILE;

    bBusy := FALSE;
    gvl_screw.bExport := FALSE; 
END_IF;*)

END_PROGRAM

// ---- NotUsedPOU/P_Error_Handling.TcPOU
PROGRAM P_Error_Handling 
VAR
	bErrorOccure	:BOOL;
	bErrorTrig		:R_trig;
	bNewSystem		:BOOL:=TRUE;

	udiStationInError				: UDINT;
	previousStationErrorCode		: UDINT;
	udiStationErrorCode				: UDINT;
	i,j,k,l,n,m: INT;
	bAlarmExist				:BOOL;
	i_current_alarm			:INT;
	j_current_alarm			: INT;
	bAlarmExist_j: BOOL;
	bAlarmExist_i: BOOL;
	b_write:BOOL;
	b_write2:BOOL;
	wstrStation :WSTRING(255);
	wstrStation2 :WSTRING(255);
	bFirstCycle				:BOOL := FALSE;
	values: ARRAY[1..175] OF INT := [
        1, 2, 3, 4, 5, 6, 7, 8, 9, 10, 11, 12, 13, 14, 15, 16, 17, 
        31, 32, 33, 34, 35, 36, 37, 38, 39, 40, 41, 42, 43, 44, 45, 
        46, 47, 48, 49, 50, 51, 52, 53, 54, 55, 56, 57, 58, 59, 60, 
        61, 62, 63, 64, 65, 66, 67, 68, 69, 70, 71, 72, 73, 74, 75, 
        76, 77, 78, 79, 84, 85, 86, 87, 88, 89, 90, 91, 92, 93, 94, 
        95, 96, 97, 98, 99, 101, 102, 103, 104, 105, 106, 107, 111, 
        112, 121, 122, 123, 124, 125, 131, 132, 141, 142, 143, 144, 
        145, 146, 147, 148, 149, 150, 151, 161, 162, 163, 164, 165, 
        171, 172, 173, 174, 175, 181, 182, 191, 192, 193, 194, 195, 
        196, 201, 202, 211, 221, 222, 223, 224, 225, 226, 227, 228, 
        229, 230, 241, 242, 243, 251, 252, 253, 254, 255, 256, 257, 
        258, 261, 262, 263, 264, 265, 266, 271, 272, 273, 281, 282, 
        283, 284, 285, 291, 292, 293, 294, 295, 296, 297, 301, 302, 
        303
    ];

	rTrigError_1:r_trig;
	bisAlarmChanged: BOOL;
END_VAR

bFirstCycle:=TRUE;
bErrorOccure			:= p_ads_1.bTrigger;
bErrorTrig				(CLK:= bErrorOccure);
//udiStationInError		:=P_ADS_ERR.udiStationInError;
IF P_ADS_ERR.udiStationInError=0 THEN
	udiStationInError:=1;
	ELSE
	udiStationInError:= P_ADS_ERR.udiStationInError;
END_IF
udiStationErrorCode:=P_ADS_ERR.udiStationErrorCode;

IF bErrorTrig.Q OR rTrigError_1.Q //AND bNewSystem 
THEN
	bAlarmExist_j:=FALSE;
	bAlarmExist_i:=FALSE;
	FOR i:=1 TO 57 DO
		 IF gvl_error.A_Error_station[i].udiStationInError 		= udiStationInError THEN
            i_current_alarm						:= i;
            bAlarmExist_i 						:= TRUE;
			gvl_error.b_empy_error:=FALSE;
			 EXIT;       
		ELSE
			gvl_error.b_empy_error:=TRUE;
			bAlarmExist_i 						:= FALSE;	
		END_IF		
	END_FOR
		FOR j:=1 TO 177 DO
		 IF gvl_error.A_Error_description[j].udiStationErrorCode 		= udiStationErrorCode THEN
            j_current_alarm						:= j;
            bAlarmExist_j 						:= TRUE;
			gvl_error.b_empy_error:=FALSE;
			previousStationErrorCode:=udiStationErrorCode;
			EXIT;
		ELSE
			gvl_error.b_empy_error:=TRUE;
			bAlarmExist_j 						:=FALSE;
            
        END_IF		
	END_FOR
		
	IF  bAlarmExist_i=TRUE AND bAlarmExist_j=TRUE THEN
        	gvl_error.ws_Stasion_In_Error				:= gvl_error.A_Error_station[i_current_alarm].wsStasionInError;
			gvl_error.udi_Station_In_Error 				:= gvl_error.A_Error_station[i_current_alarm].udiStationInError ;
			gvl_error.udi_Station_In_Error_Code 		:= gvl_error.A_Error_description[j_current_alarm].udiStationErrorCode ;
			gvl_error.ws_Station_Error_Description		:= gvl_error.A_Error_description[j_current_alarm].wsStationErrorDescription;
			gvl_error.ws_Station_Error_Description_2 	:= P_ADS_ERR.sStationErrorDescription2;
    	ELSE
		i_current_alarm := 0;
		gvl_error.b_empy_error:=TRUE;
	END_IF
	
END_IF

gvl_error.b_new_system:=bNewSystem;

IF bFirstCycle=TRUE OR b_write=TRUE THEN
	gvl_error.A_Error_station[1].udiStationInError:=1;
	gvl_error.A_Error_station[1].wsStasionInError:="Station1";
	gvl_error.A_Error_description[176].udiStationErrorCode:=311;
	gvl_error.A_Error_description[176].wsStationErrorDescription:="Error176";
	gvl_error.A_Error_description[177].udiStationErrorCode:=18;
	gvl_error.A_Error_description[177].wsStationErrorDescription:="Error177";
	
	FOR k := 2 TO 57 DO
    gvl_error.A_Error_station[k].udiStationInError := 9 + k; // udiStationInError od 11 do 66
    
    wstrStation := WCONCAT("Station", INT_TO_WSTRING(k));
    gvl_error.A_Error_station[k].wsStasionInError := wstrStation;  // Przypisanie wartości WSTRING
	END_FOR
	FOR l := 1 TO 175 DO
    
    wstrStation2 := WCONCAT("Error", INT_TO_WSTRING(l));
    gvl_error.A_Error_description[l].wsStationErrorDescription := wstrStation2;  // Przypisanie wartości WSTRING
	END_FOR
END_IF

IF bFirstCycle=TRUE OR b_write2=TRUE	THEN
	m := 1;  // Inicjalizacja indeksu dla tablicy values
	FOR n := 1 TO 175 DO
    gvl_error.A_Error_description[n].udiStationErrorCode := values[m];  // Przypisanie wartości z tablicy values do A_Error_description
    m := m + 1;  // Przejście do następnej wartości
	END_FOR	

END_IF

IF (previousStationErrorCode <> udiStationErrorCode) AND (udiStationErrorCode <>0)  THEN
	bisAlarmChanged:=TRUE;
END_IF
IF(previousStationErrorCode = udiStationErrorCode) THEN
		bisAlarmChanged:=FALSE;
END_IF
	rTrigError_1(CLK:=bisAlarmChanged);
gvl_error.b_empy_error:=FALSE;

END_PROGRAM
